// TIA Portal V19 export
TYPE "LAF_typeJobsCommands"
TITLE = LAF_typeJobCommands
// Commands related to job select
// stored: Access Published
   STRUCT
      setJobNumber : DInt;   // Number of the job to be executed
      reset : Bool;   // Reset all jobs
   END_STRUCT;
END_TYPE
